// TIA Portal V19 export
FUNCTION_BLOCK "VFD Type"   // FB9, LAD
{ S7_Optimized_Access := 'TRUE' }
// stored: MemoryReserve 100, SetENOAutomatically false
   VAR_INPUT
      Overload_IN { ExternalAccessible := 'False'; ExternalVisible := 'False'; ExternalWritable := 'False'} : Bool;
      Isolator_in { ExternalAccessible := 'False'; ExternalVisible := 'False'; ExternalWritable := 'False'} : Bool;
      "Motor Number" : Int;
      HWIDSTW { ExternalAccessible := 'False'; ExternalVisible := 'False'; ExternalWritable := 'False'} : HW_IO;
      HWIDZSSW { ExternalAccessible := 'False'; ExternalVisible := 'False'; ExternalWritable := 'False'} : HW_IO;
      "POPUP NUmber" : Int;
      "Auto Run" : Bool;
      "Auto Speed" : Real;
      "Ack Error" : Bool;
      Ref_Speed { ExternalAccessible := 'False'; ExternalVisible := 'False'; ExternalWritable := 'False'} : Real;
      Ref_Current : Real;
      Ref_Torque { ExternalAccessible := 'False'; ExternalVisible := 'False'; ExternalWritable := 'False'} : Real;
   END_VAR
   VAR_OUTPUT
      "Drive Running" : Bool;
      "Actual Speed" : Real;
      Axis_Active : Bool;
      Lockout_Active : Bool;
      Error_Present : Bool;
      VFD_Fault : Int;
      "Motor State" : Int;
      Act_Current : Real;
      Act_torque : Real;
   END_VAR
   VAR_IN_OUT
      drive_status { ExternalAccessible := 'False'; ExternalVisible := 'False'; ExternalWritable := 'False'} : Word;
   END_VAR
   VAR
      Speed_SP : Real;
      "Sts Running" : Bool;
   END_VAR
   VAR RETAIN
      IEC_Counter_0_Instance { ExternalAccessible := 'False'; ExternalVisible := 'False'; ExternalWritable := 'False'} : CTU_INT;
   END_VAR
   VAR
      "SCALED sp" : Real;
      "speed to drive" : Real;
      Speed_From_Drive : Real;
      "SCALED sp_1" : Real;
   END_VAR
BEGIN

REGION Network 1
   // Refspeed = p2000, ref_Current = P2002, Ref_torque = P2003
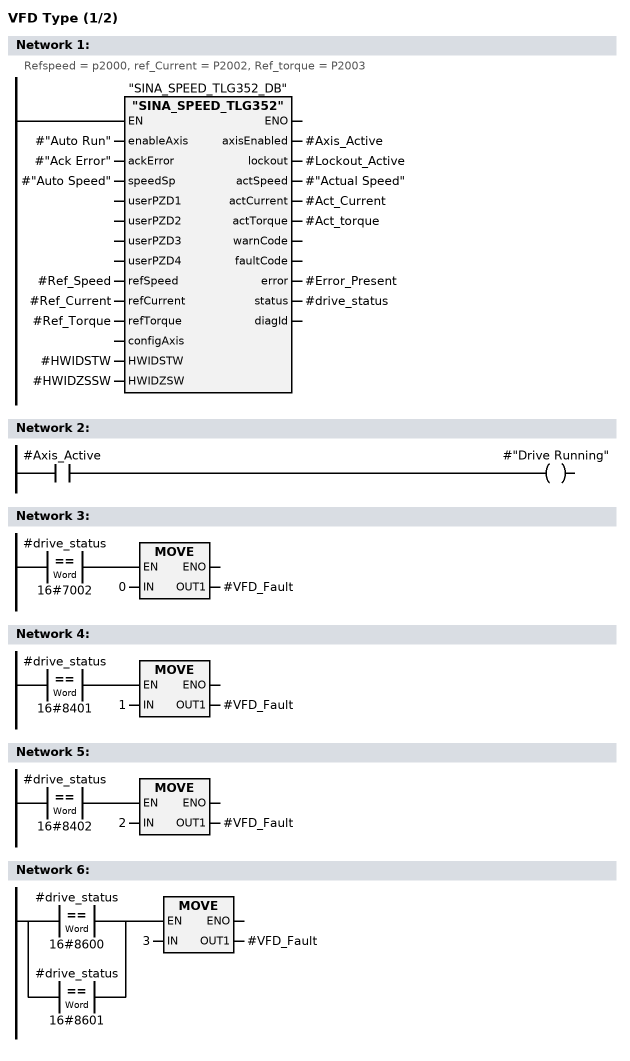
   RUNG wire#powerrail
      "SINA_SPEED_TLG352_DB"(enableAxis := #"Auto Run", ackError := #"Ack Error", speedSp := #"Auto Speed", userPZD1 :=, userPZD2 :=, userPZD3 :=, userPZD4 :=, refSpeed := #Ref_Speed, refCurrent := #Ref_Current, refTorque := #Ref_Torque, configAxis :=, HWIDSTW := #HWIDSTW, HWIDZSW := #HWIDZSSW, axisEnabled => #Axis_Active, lockout => #Lockout_Active, actSpeed => #"Actual Speed", actCurrent => #Act_Current, actTorque => #Act_torque, warnCode =>, faultCode =>, error => #Error_Present, status => #drive_status, diagId =>)
   END_RUNG
   // the same network as SCL:
   "SINA_SPEED_TLG352_DB"(enableAxis := #"Auto Run",   // "SINA_SPEED_TLG352"
                          ackError := #"Ack Error",
                          speedSp := #"Auto Speed",
                          refSpeed := #Ref_Speed,
                          refCurrent := #Ref_Current,
                          refTorque := #Ref_Torque,
                          HWIDSTW := #HWIDSTW,
                          HWIDZSW := #HWIDZSSW,
                          axisEnabled => #Axis_Active,
                          lockout => #Lockout_Active,
                          actSpeed => #"Actual Speed",
                          actCurrent => #Act_Current,
                          actTorque => #Act_torque,
                          error => #Error_Present,
                          status => #drive_status);
END_REGION

REGION Network 2
   RUNG wire#powerrail
      Contact( #Axis_Active )
      Coil( #"Drive Running" )
   END_RUNG
   // the same network as SCL:
   #"Drive Running" := #Axis_Active;
END_REGION

REGION Network 3
   RUNG wire#powerrail
      { S7_Templates := "SrcType := Word" } EQ_Contact(in1 := #drive_status, in2 := 16#7002)
      Move(in := 0, out1 => #VFD_Fault)
   END_RUNG
   // the same network as SCL:
   IF #drive_status = 16#7002 THEN #VFD_Fault := 0; END_IF;
END_REGION

REGION Network 4
   RUNG wire#powerrail
      { S7_Templates := "SrcType := Word" } EQ_Contact(in1 := #drive_status, in2 := 16#8401)
      Move(in := 1, out1 => #VFD_Fault)
   END_RUNG
   // the same network as SCL:
   IF #drive_status = 16#8401 THEN #VFD_Fault := 1; END_IF;
END_REGION

REGION Network 5
   RUNG wire#powerrail
      { S7_Templates := "SrcType := Word" } EQ_Contact(in1 := #drive_status, in2 := 16#8402)
      Move(in := 2, out1 => #VFD_Fault)
   END_RUNG
   // the same network as SCL:
   IF #drive_status = 16#8402 THEN #VFD_Fault := 2; END_IF;
END_REGION

REGION Network 6
   RUNG wire#powerrail
      { S7_Templates := "SrcType := Word" } EQ_Contact(in1 := #drive_status, in2 := 16#8600)
      wire#w1
      Move(in := 3, out1 => #VFD_Fault)
   END_RUNG
   RUNG wire#powerrail
      { S7_Templates := "SrcType := Word" } EQ_Contact(in1 := #drive_status, in2 := 16#8601)
   END_RUNG wire#w1
   // the same network as SCL:
   IF (#drive_status = 16#8600) OR (#drive_status = 16#8601) THEN #VFD_Fault := 3; END_IF;
END_REGION

REGION Network 7
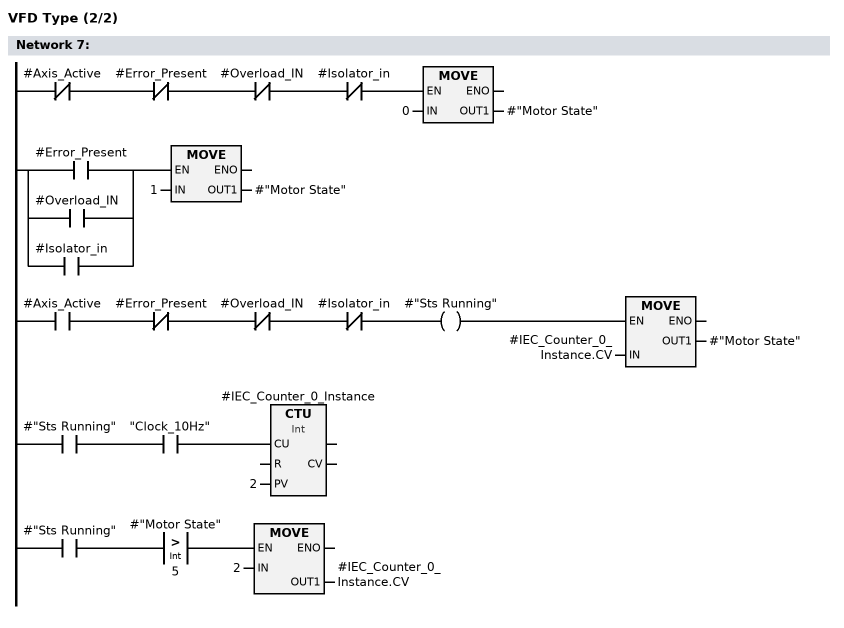
   RUNG wire#powerrail
      I_Contact( #Axis_Active )
      I_Contact( #Error_Present )
      I_Contact( #Overload_IN )
      I_Contact( #Isolator_in )
      Move(in := 0, out1 => #"Motor State")
   END_RUNG
   RUNG wire#powerrail
      Contact( #Error_Present )
      wire#w1
      Move(in := 1, out1 => #"Motor State")
   END_RUNG
   RUNG wire#powerrail
      Contact( #Overload_IN )
   END_RUNG wire#w1
   RUNG wire#powerrail
      Contact( #Isolator_in )
   END_RUNG wire#w1
   RUNG wire#powerrail
      Contact( #Axis_Active )
      I_Contact( #Error_Present )
      I_Contact( #Overload_IN )
      I_Contact( #Isolator_in )
      Coil( #"Sts Running" )
      Move(in := #IEC_Counter_0_Instance.CV, out1 => #"Motor State")
   END_RUNG
   RUNG wire#powerrail
      Contact( #"Sts Running" )
      Contact( "Clock_10Hz" )
      { S7_Templates := "value_type := Int" } #IEC_Counter_0_Instance.CTU(r :=, pv := 2, cv =>)
   END_RUNG
   RUNG wire#powerrail
      Contact( #"Sts Running" )
      { S7_Templates := "SrcType := Int" } GT_Contact(in1 := #"Motor State", in2 := 5)
      Move(in := 2, out1 => #IEC_Counter_0_Instance.CV)
   END_RUNG
   // the same network as SCL:
   IF NOT #Axis_Active AND NOT #Error_Present AND NOT #Overload_IN AND NOT #Isolator_in THEN
       #"Motor State" := 0;
   END_IF;
   IF #Error_Present OR #Overload_IN OR #Isolator_in THEN #"Motor State" := 1; END_IF;
   #"Sts Running" := #Axis_Active AND NOT #Error_Present AND NOT #Overload_IN AND NOT #Isolator_in;
   IF #"Sts Running" THEN #"Motor State" := #IEC_Counter_0_Instance.CV; END_IF;
   #IEC_Counter_0_Instance(CU := #"Sts Running" AND "Clock_10Hz", PV := 2);   // CTU
   IF #"Sts Running" AND (#"Motor State" > 5) THEN #IEC_Counter_0_Instance.CV := 2; END_IF;
END_REGION
END_FUNCTION_BLOCK
